# EPICS autosave request: iocBoot/iocUSB1608G-2AO/auto_settings.req
file "USB1608G_2AO_settings.req", P=$(P)
